INTERFACE IInspector EXTENDS __SYSTEM.IQueryInterface

PROPERTY Busy : BOOL
GET
END_GET
END_PROPERTY

(*~
	<docu>
		<summary>
			Gets common data settings of inspectors.
		</summary>			
	</docu>	
~*)
PROPERTY CommonData : REFERENCE TO TcoInspectorData
GET
END_GET
END_PROPERTY

PROPERTY Coordinator : TcoCore.ITcoCoordinator
GET
END_GET
END_PROPERTY

PROPERTY Done : BOOL
GET
END_GET
END_PROPERTY

METHOD HideOverride : IInspector
END_METHOD

METHOD HideRetry : IInspector
END_METHOD

METHOD HideTerminate : IInspector
END_METHOD

PROPERTY Identity : ULINT
GET
END_GET
END_PROPERTY

METHOD Instruct : IInspector
VAR_INPUT
	inInstruction:STRING(255);
END_VAR
END_METHOD

METHOD InstructWithImage : IInspector
VAR_INPUT
	inImageSource:STRING(255);
	inHeight:REAL;
	inWidth:REAL;
END_VAR
END_METHOD

METHOD OnFail : IOnFail
END_METHOD

PROPERTY OverInspected : BOOL
GET
END_GET
END_PROPERTY

PROPERTY Result : eInspectorResult
GET
END_GET
END_PROPERTY

(*~
	<docu>
		<summary>
			Updates comprehensive result. The comprehensive result is set to `Failed` when any inspection fails or is inconclusive.
			Any bypassed or excluded inspection are not taken in the account.			
		</summary>			
	</docu>	
~*)
METHOD UpdateComprehensiveResult : IInspector
VAR_IN_OUT
	(*~
	<docu>
		<summary>
			Comprehensive result data structure to be updated.	
		</summary>			
	</docu>	
	~*)
    inoResult : TcoComprehensiveResult;
END_VAR
END_METHOD

(*~
	<docu>
		<summary>
			Provide information about the Inspector name (if there are multiple inspectors, only the failed ones will be displayed).  (e.g. {attribute addProperty Name "Bolt presence inspection"})
		</summary>			
	</docu>	
~*)
METHOD WithDescription : IInspector
END_METHOD

(*~
	<docu>
		<summary>
			Provide information about ErrorCode (if there are multiple inspectors, only the failed ones will be displayed). Error codes shoud be defined in Inspectors
		</summary>			
	</docu>	
~*)
METHOD WithErrorCode : IInspector
END_METHOD

(*~
	<docu>
		<summary>
			Provide information about Failure Description (if there are multiple inspectors, only the failed ones will be displayed). Failure description shoud be defined in Inspectors.
		</summary>			
	</docu>	
~*)
METHOD WithFailureDescription : IInspector
END_METHOD

END_INTERFACE

(* stored: Version 1.1.0.1, ProductVersion 3.1.4024.12
   Itf IInspector: Id {0cbe9e39-d5a4-05af-17ce-7965efd20de3}
   Property Busy: Id {b32bf15d-c374-0d51-2e79-45bad14701d4}
   Get Get: Id {ebd05d89-2b98-0f79-0951-70a8ea77ee5c}
   Property CommonData: Id {042544e7-f282-06f0-051b-e2f8bd92dc63}
   Get Get: Id {9b5ef77f-71b0-07b1-3bad-27c8bab87325}
   Property Coordinator: Id {53464262-388f-0508-055a-3695c0743081}
   Get Get: Id {e54c0b21-129c-0276-1867-e027cd67689d}
   Property Done: Id {619d20fa-40bc-0c73-013c-9ce9a7b16b05}
   Get Get: Id {dda1cead-ae16-0ba2-2984-226a50200b84}
   Method HideOverride: Id {b431c33c-95f9-04d3-2b46-90c0ee1194d0}
   Method HideRetry: Id {d3a6b912-afba-0dc7-214b-0768c024db38}
   Method HideTerminate: Id {1fdd4937-bf43-037d-3d7e-7880941def25}
   Property Identity: Id {30ca9dd1-1e56-01cf-3dbc-58c99beb7408}
   Get Get: Id {275ba232-6810-0478-08ce-630296e4e874}
   Method Instruct: Id {224318fe-b0d5-052c-0281-f5490a547cae}
   Method InstructWithImage: Id {27b2b815-048c-0e70-370e-3cb41b72265b}
   Method OnFail: Id {ac3abd9c-363c-070f-178a-504f9b7741ff}
   Property OverInspected: Id {8def8039-9580-0717-1f67-557c2ea921c0}
   Get Get: Id {7ec14b78-0f82-0a30-2aad-7349dddb37bc}
   Property Result: Id {059b95a9-368b-016b-1e77-bc829a9a2a15}
   Get Get: Id {11bcb09e-df05-0600-3fcc-c1e8eab49bfc}
   Method UpdateComprehensiveResult: Id {91a1c4e6-d695-0902-3533-5110a9d88e30}
   Method WithDescription: Id {f186ff2b-9fb3-02e9-3cf4-5ab10df77bbe}
   Method WithErrorCode: Id {9309859b-94bb-06e6-10ab-dfe20f9fd755}
   Method WithFailureDescription: Id {2d34164d-c11f-0306-2984-768b8e4e972b} *)
